// Mitsubishi GX Works2 project: 07091초에10카운트100까지   PLC: Q02/Q02H

PROGRAM MAIN
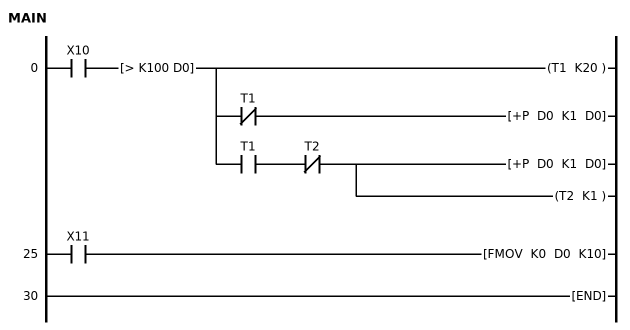
0     LD      X10
      AND>    K100 D0
      OUT     T1 K20
      MPS
      ANI     T1
      +P      D0 K1 D0
      MPP
      AND     T1
      ANI     T2
      +P      D0 K1 D0
      OUT     T2 K1
25    LD      X11
      FMOV    K0 D0 K10
30    END
END_PROGRAM
